Yaskawa INFORM job: GO-START.JBI

/JOB
//NAME GO-START
///FOLDERNAME FOLDER001
//POS
///NPOS 0,0,0,1,0,0
///TOOL 1
///POSTYPE ROBOT
///RECTAN
///RCONF 0,0,0,0,0,0,0,0,0,0,0,0,0,0,0,0,0,0,0,0,0,0,0,0
P00090=1011.893,162.000,653.762,180.0000,-45.0000,0.0000
//INST
///DATE 2025/09/30 16:23
///ATTR SC,RW
///GROUP1 RB1
NOP
MOVJ P090 VJ=100.00 PL=3
END
